RoboDK station: CollisionSimulation_Welding Station - Fanuc.rdk

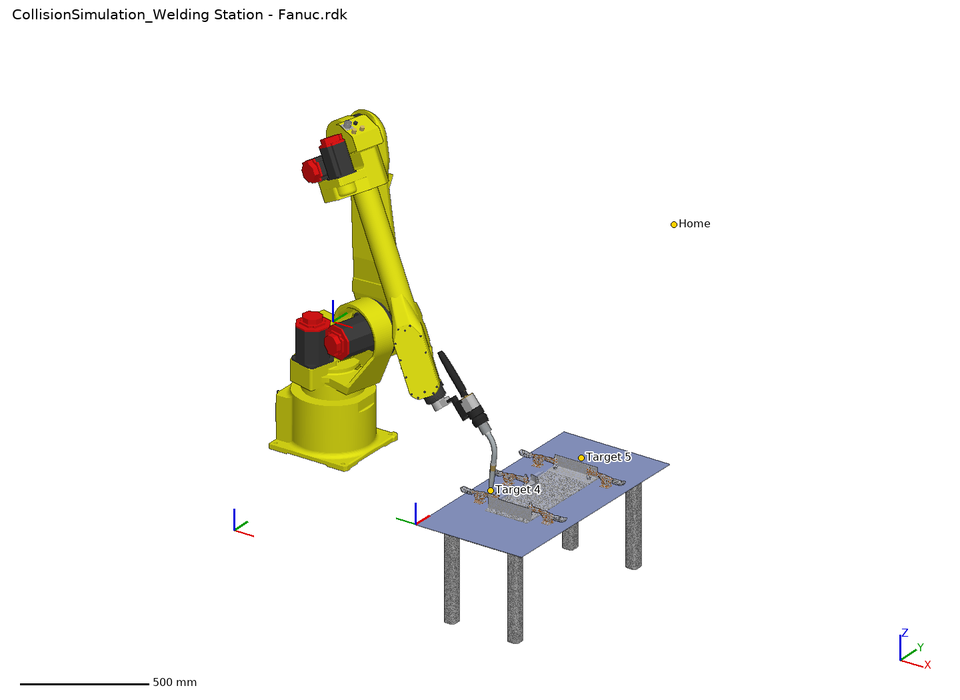
[picture v0: the station drawn from its stored meshes, robots at their saved joint values, targets as dots, program paths as lines]
Station CollisionSimulation_Welding Station - Fanuc (saved by RoboDK 5.2.5). Poses are relative to the parent item; angles as X-Y-Z fixed-axis rotations.
Station parameters (name, value as stored): Torch1, 4, red, 0, OPC-UA, opc.tcp://localhost:4840, CollisionFreePlanner, Fanuc ARC Mate 120iB/10L, CollisionFreePlanner-Rob Fanuc ARC Mate 120iB/10L
  - frame Fanuc ARC Mate 120iB/10L Base at (0, 0, 525) mm
    - robot Fanuc ARC Mate 120iB/10L: 6 axes, payload 10 kg, reach 1885 mm, repeatability 0.1 mm, weight 225 kg
        modified DH rows (alpha deg, a mm, theta deg, d mm): 0, 0, 0, 525; -90, 150, -90, 0; 0, 770, 0, 0; -90, 100, 0, 960; 90, 0, 0, 0; -90, 0, 0, 100
        base shift (0, 0, -525) mm
        joint limits [-20, -50, -170, -200, -140, -150] to [51, 150, 250, 200, 140, 450]; home [0, 0, 0, 0, 0, 0]; saved at [-14.441, -10.288, -62.244, 43.223, 13.017, -31.04]
      - tool Daihen OTC weld gun, TCP at (-2, 0, 402) mm, rotated rx 0 ry 45 rz 180 deg, size 201.6 x 65.1 x 567.7 mm
  - frame Table at (741.65, -500, 58.58) mm, rotated rx 0 ry 0 rz 90 deg
    - target Home (joint target) at (500, -870.35, 1334.42) mm, rotated rx -180 ry 45 rz 90 deg; joints [0, 0, 0, 0, 0, 0] of Fanuc ARC Mate 120iB/10L
    - object Weld 1 at (0, 0, 0) mm, size 1000 x 500 x 492.1 mm, geometry from Weld 1.step
    - target Target 4 (Cartesian target) at (363.32, -98.01, 25.38) mm, rotated rx -180 ry -6.79 rz 90 deg; joints [-14.441, -10.288, -62.244, 43.223, 13.017, -31.04] of Fanuc ARC Mate 120iB/10L
    - target Target 5 (Cartesian target) at (749.74, -256.93, 58.5) mm, rotated rx -180 ry -6.79 rz 90 deg; joints [19.906, 1.322, -60.065, -62.022, 13.796, 45.438] of Fanuc ARC Mate 120iB/10L
  - frame World at (-304.32, -233.92, -366.75) mm
  - object box at (0, 0, 0) mm, size 100 x 100 x 100 mm, geometry from box.sld
  - program Target4ToTarget5 (10 instructions, listed below)
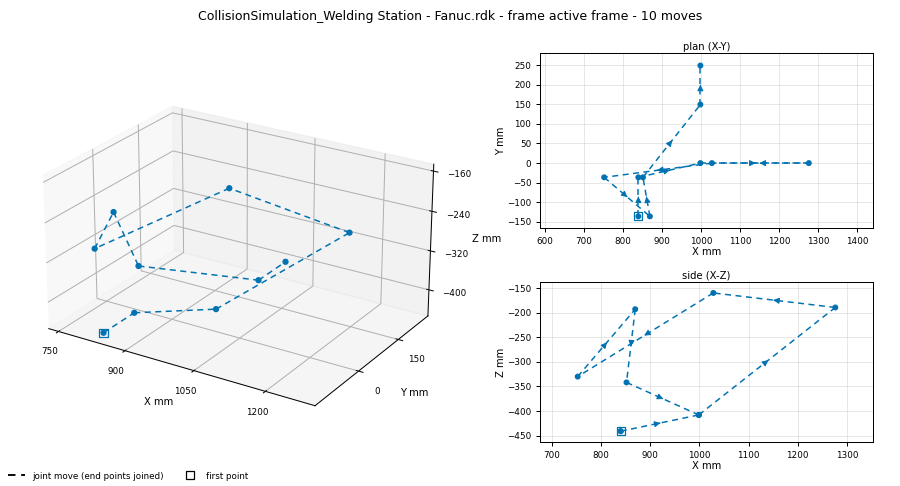
[picture p0: tool path of CollisionSimulation_Welding Station - Fanuc.rdk in frame active frame, 10 of 10 moves have a stored position in this frame; points joined in program order, loops and branches not executed]

--- program Target4ToTarget5 (robot Fanuc ARC Mate 120iB/10L) ---
  MoveJ (Pt 1 (S48)) to (839.66, -136.68, -441.04) mm, rotated rx -180 ry -6.79 rz 180 deg; joints [-14.441, -10.288, -62.244, 43.223, 13.017, -31.04]
  MoveJ (Pt 2 (S26)) to (839.66, -36.68, -441.04) mm, rotated rx -180 ry -6.79 rz 180 deg; joints [-3.953, -12.01, -61.768, 13.927, 10.205, -10.607]
  MoveJ (Pt 3 (S21)) to (998.59, -0.26, -407.92) mm, rotated rx -180 ry -6.79 rz 180 deg; joints [-0.022, -1.965, -60.04, 0.093, 8.249, -0.075]
  MoveJ (Pt 4 (S25)) to (1276.4, -0.26, -189.24) mm, rotated rx -180 ry -6.79 rz 180 deg; joints [-0.015, 2.483, -41.617, -0.054, -10.174, 0.065]
  MoveJ (Pt 5 (S38)) to (1028.15, -0.26, -159.68) mm, rotated rx -180 ry -6.79 rz 180 deg; joints [-0.021, -20.043, -36.273, -0.048, -15.518, 0.062]
  MoveJ (Pt 6 (S45)) to (752.19, -36.68, -329.92) mm, rotated rx -180 ry -6.79 rz 180 deg; joints [-4.73, -44.724, -35.859, -10.479, -16.285, 13.787]
  MoveJ (Pt 7 (S49)) to (869.23, -136.68, -192.8) mm, rotated rx -180 ry -6.79 rz 180 deg; joints [-13.709, -34.558, -32.485, -23.317, -21.736, 32.67]
  MoveJ (Pt 8 (S29)) to (851.49, -36.67, -341.74) mm, rotated rx 180 ry -6.79 rz -180 deg; joints [-3.867, -24.972, -47.806, -30.593, -4.702, 33.549]
  MoveJ (Pt 9 (S11)) to (998.59, 149.74, -407.92) mm, rotated rx -180 ry -6.79 rz 180 deg; joints [12.25, -0.729, -60.08, -44.846, 10.725, 34.66]
  MoveJ (Pt 10 (S6)) to (998.59, 249.74, -407.92) mm, rotated rx -180 ry -6.79 rz 180 deg; joints [19.906, 1.322, -60.065, -62.022, 13.796, 45.438]
